ABB RAPID module: MovementChech_5abb.mod

MODULE MainModule
    TASK PERS tooldata tool1 := [
    TRUE,
    [[3.25653, -2.2499, 106.27], [1, 0, 0, 0]],
    [0.2, [0, 0, 50], [1, 0, 0, 0], 0, 0, 0]
    ];

    PERS robtarget p_home := [
    [342.30, -38.16, 327.52],
    [1.20614E-05, 0.456804, -0.889567, -5.42704E-06],
    [-1, -1, -1, 0],
    [9E+09, 9E+09, 9E+09, 9E+09, 9E+09, 9E+09]
    ];

    PERS robtarget p_assembly := [
    [342.30, -38.16, 327.52],
    [1.20614E-05, 0.456804, -0.889567, -5.42704E-06],
    [-1, -1, -1, 0],
    [9E+09, 9E+09, 9E+09, 9E+09, 9E+09, 9E+09]
    ];

    PERS robtarget p_axle_pickup := [
    [342.30, -38.16, 327.52],
    [1.20614E-05, 0.456804, -0.889567, -5.42704E-06],
    [-1, -1, -1, 0],
    [9E+09, 9E+09, 9E+09, 9E+09, 9E+09, 9E+09]
    ];

    PERS robtarget p_axle_pickdown := [
    [342.30, -38.16, 327.52],
    [1.20614E-05, 0.456804, -0.889567, -5.42704E-06],
    [-1, -1, -1, 0],
    [9E+09, 9E+09, 9E+09, 9E+09, 9E+09, 9E+09]
    ];

    PERS robtarget p_axle_assem_up := [
    [342.30, -38.16, 327.52],
    [1.20614E-05, 0.456804, -0.889567, -5.42704E-06],
    [-1, -1, -1, 0],
    [9E+09, 9E+09, 9E+09, 9E+09, 9E+09, 9E+09]
    ];

    PERS robtarget p_axle_assem_down := [
    [342.30, -38.16, 327.52],
    [1.20614E-05, 0.456804, -0.889567, -5.42704E-06],
    [-1, -1, -1, 0],
    [9E+09, 9E+09, 9E+09, 9E+09, 9E+09, 9E+09]
    ];

    PERS robtarget p_tier_up := [
    [342.30, -38.16, 327.52],
    [1.20614E-05, 0.456804, -0.889567, -5.42704E-06],
    [-1, -1, -1, 0],
    [9E+09, 9E+09, 9E+09, 9E+09, 9E+09, 9E+09]
    ];

    PERS robtarget p_tier_down := [
    [342.30, -38.16, 327.52],
    [1.20614E-05, 0.456804, -0.889567, -5.42704E-06],
    [-1, -1, -1, 0],
    [9E+09, 9E+09, 9E+09, 9E+09, 9E+09, 9E+09]
    ];

    PERS robtarget p_tier_link_1 := [
    [342.30, -38.16, 327.52],
    [1.20614E-05, 0.456804, -0.889567, -5.42704E-06],
    [-1, -1, -1, 0],
    [9E+09, 9E+09, 9E+09, 9E+09, 9E+09, 9E+09]
    ];

    PERS robtarget p_tier_link_1_down := [
    [342.30, -38.16, 327.52],
    [1.20614E-05, 0.456804, -0.889567, -5.42704E-06],
    [-1, -1, -1, 0],
    [9E+09, 9E+09, 9E+09, 9E+09, 9E+09, 9E+09]
    ];

    PERS robtarget p_tier_link_2 := [
    [342.30, -38.16, 327.52],
    [1.20614E-05, 0.456804, -0.889567, -5.42704E-06],
    [-1, -1, -1, 0],
    [9E+09, 9E+09, 9E+09, 9E+09, 9E+09, 9E+09]
    ];

    PERS robtarget p_tier_link_2_down := [
    [342.30, -38.16, 327.52],
    [1.20614E-05, 0.456804, -0.889567, -5.42704E-06],
    [-1, -1, -1, 0],
    [9E+09, 9E+09, 9E+09, 9E+09, 9E+09, 9E+09]
    ];

    PERS robtarget p_tier_link_3 := [
    [342.30, -38.16, 327.52],
    [1.20614E-05, 0.456804, -0.889567, -5.42704E-06],
    [-1, -1, -1, 0],
    [9E+09, 9E+09, 9E+09, 9E+09, 9E+09, 9E+09]
    ];

    PERS robtarget p_tier_link_3_down := [
    [342.30, -38.16, 327.52],
    [1.20614E-05, 0.456804, -0.889567, -5.42704E-06],
    [-1, -1, -1, 0],
    [9E+09, 9E+09, 9E+09, 9E+09, 9E+09, 9E+09]
    ];

    PERS robtarget p_tier_link_4 := [
    [342.30, -38.16, 327.52],
    [1.20614E-05, 0.456804, -0.889567, -5.42704E-06],
    [-1, -1, -1, 0],
    [9E+09, 9E+09, 9E+09, 9E+09, 9E+09, 9E+09]
    ];

    PERS robtarget p_tier_link_4_down := [
    [342.30, -38.16, 327.52],
    [1.20614E-05, 0.456804, -0.889567, -5.42704E-06],
    [-1, -1, -1, 0],
    [9E+09, 9E+09, 9E+09, 9E+09, 9E+09, 9E+09]
    ];

    ! ===== Lower body station (chassis supply location) =====
    ! ===== 하부체 스테이션 (차체 하부 공급 위치) =====
    PERS robtarget p_Lower_body_pickup := [
    [342.30, -38.16, 327.52],
    [1.20614E-05, 0.456804, -0.889567, -5.42704E-06],
    [-1, -1, -1, 0],
    [9E+09, 9E+09, 9E+09, 9E+09, 9E+09, 9E+09]
    ];

    PERS robtarget p_Lower_body_pickdown := [
    [342.30, -38.16, 327.52],
    [1.20614E-05, 0.456804, -0.889567, -5.42704E-06],
    [-1, -1, -1, 0],
    [9E+09, 9E+09, 9E+09, 9E+09, 9E+09, 9E+09]
    ];

    PERS robtarget p_Lower_body_link := [
    [342.30, -38.16, 327.52],
    [1.20614E-05, 0.456804, -0.889567, -5.42704E-06],
    [-1, -1, -1, 0],
    [9E+09, 9E+09, 9E+09, 9E+09, 9E+09, 9E+09]
    ];

    PERS robtarget p_Lower_body_link_down := [
    [342.30, -38.16, 327.52],
    [1.20614E-05, 0.456804, -0.889567, -5.42704E-06],
    [-1, -1, -1, 0],
    [9E+09, 9E+09, 9E+09, 9E+09, 9E+09, 9E+09]
    ];

    ! ===== Battery station (battery supply location) =====
    ! ===== 배터리 스테이션 (배터리 공급 위치) =====
    PERS robtarget p_battery_pickup := [
    [342.30, -38.16, 327.52],
    [1.20614E-05, 0.456804, -0.889567, -5.42704E-06],
    [-1, -1, -1, 0],
    [9E+09, 9E+09, 9E+09, 9E+09, 9E+09, 9E+09]
    ];

    PERS robtarget p_battery_pickdown := [
    [342.30, -38.16, 327.52],
    [1.20614E-05, 0.456804, -0.889567, -5.42704E-06],
    [-1, -1, -1, 0],
    [9E+09, 9E+09, 9E+09, 9E+09, 9E+09, 9E+09]
    ];

    PERS robtarget p_battery_link_up := [
    [342.30, -38.16, 327.52],
    [1.20614E-05, 0.456804, -0.889567, -5.42704E-06],
    [-1, -1, -1, 0],
    [9E+09, 9E+09, 9E+09, 9E+09, 9E+09, 9E+09]
    ];

    PERS robtarget p_battery_link_down := [
    [342.30, -38.16, 327.52],
    [1.20614E-05, 0.456804, -0.889567, -5.42704E-06],
    [-1, -1, -1, 0],
    [9E+09, 9E+09, 9E+09, 9E+09, 9E+09, 9E+09]
    ];

    ! ===== Motor station - NOT used in Run_Assembly_Cycle yet (out of scope for now) =====
    ! ===== 모터 스테이션 - 아직 Run_Assembly_Cycle에서 사용 안 함 (현재 작업 범위 밖) =====
    PERS robtarget p_motor_pickup := [
    [342.30, -38.16, 327.52],
    [1.20614E-05, 0.456804, -0.889567, -5.42704E-06],
    [-1, -1, -1, 0],
    [9E+09, 9E+09, 9E+09, 9E+09, 9E+09, 9E+09]
    ];

    PERS robtarget p_motor_pickdown := [
    [342.30, -38.16, 327.52],
    [1.20614E-05, 0.456804, -0.889567, -5.42704E-06],
    [-1, -1, -1, 0],
    [9E+09, 9E+09, 9E+09, 9E+09, 9E+09, 9E+09]
    ];

    PERS robtarget p_motor_linkup := [
    [342.30, -38.16, 327.52],
    [1.20614E-05, 0.456804, -0.889567, -5.42704E-06],
    [-1, -1, -1, 0],
    [9E+09, 9E+09, 9E+09, 9E+09, 9E+09, 9E+09]
    ];

    PERS robtarget p_motor_linkdown := [
    [342.30, -38.16, 327.52],
    [1.20614E-05, 0.456804, -0.889567, -5.42704E-06],
    [-1, -1, -1, 0],
    [9E+09, 9E+09, 9E+09, 9E+09, 9E+09, 9E+09]
    ];

    PERS robtarget p_assembly_pickup := [
    [342.30, -38.16, 327.52],
    [1.20614E-05, 0.456804, -0.889567, -5.42704E-06],
    [-1, -1, -1, 0],
    [9E+09, 9E+09, 9E+09, 9E+09, 9E+09, 9E+09]
    ];

    PERS robtarget p_assembly_pickdown := [
    [342.30, -38.16, 327.52],
    [1.20614E-05, 0.456804, -0.889567, -5.42704E-06],
    [-1, -1, -1, 0],
    [9E+09, 9E+09, 9E+09, 9E+09, 9E+09, 9E+09]
    ];

    ! ===== Exit conveyor =====
    ! ===== 출하 컨베이어 =====
    PERS robtarget p_conveyor_Exit_up := [
    [342.30, -38.16, 327.52],
    [1.20614E-05, 0.456804, -0.889567, -5.42704E-06],
    [-1, -1, -1, 0],
    [9E+09, 9E+09, 9E+09, 9E+09, 9E+09, 9E+09]
    ];

    PERS robtarget p_conveyor_Exit_down := [
    [342.30, -38.16, 327.52],
    [1.20614E-05, 0.456804, -0.889567, -5.42704E-06],
    [-1, -1, -1, 0],
    [9E+09, 9E+09, 9E+09, 9E+09, 9E+09, 9E+09]
    ];


    PROC Main()
        MoveL p_home, v150, fine, tool1;

        ! Axle
        MoveJ p_axle_pickup, v_fast, z30, tool1;
        MoveL p_axle_pickdown, v_slow, fine, tool1;
        Grip_On;
        SetDO do05_Axle_Cylinder_Forward, 0;
        MoveL p_axle_pickup, v_slow, fine, tool1;

        MoveL p_assembly, v_fast, z30, tool1;
        MoveL p_axle_assem_up, v_fast, z30, tool1;
        MoveL p_axle_assem_down, v_slow, fine, tool1;
        SetDO do07_Axle_Gripper_On, 1;
        Grip_Off;
        MoveL p_axle_assem_up, v_slow, fine, tool1;

        ! Lower_body
        MoveJ p_Lower_body_pickup, v_fast, z30, tool1;
        MoveL p_Lower_body_pickdown, v_slow, fine, tool1;
        Grip_On;
        MoveL p_Lower_body_pickup, v_slow, fine, tool1;

        MoveL p_assembly, v_fast, z30, tool1;
        MoveL p_Lower_body_link, v_fast, z30, tool1;
        MoveL p_Lower_body_link_down, v_slow, fine, tool1;
        Grip_Off;
        MoveL p_Lower_body_link, v_slow, fine, tool1;

        !Battery
        MoveL p_battery_pickup, v_fast, z30, tool1;
        MoveL p_battery_pickdown, v_slow, fine, tool1;
        Grip_On;
        MoveL p_battery_pickup, v_fast, fine, tool1;

        MoveL p_assembly, v_fast, z30, tool1;
        MoveL p_battery_link_up, v_fast, z30, tool1;
        MoveL p_battery_link_down, v_slow, fine, tool1;
        Grip_Off;
        MoveL p_battery_link_up, v_slow, fine, tool1;

        !
    ENDPROC

    PROC Grip_On()
        PulseDO \PLength := 0.2, do00_grip_on;
        WaitDI di00_grip_on_sen, 1;
        WaitTime 0.1;
    ENDPROC

    PROC Grip_Off()
        PulseDO \PLength := 0.2, do01_grip_off;
        WaitDI di01_grip_off_sen, 1;
        WaitTime 0.1;
    ENDPROC

ENDMODULE
